{attribute 'qualified_only'}
VAR_GLOBAL
	senNO				: FB_Sensor_NO;
	senNC				: FB_Sensor_NC;
	senNO_2inRow		: FB_Sensor_NO_2InRow;
	
	senNO_TestDecorator			: FB_Sensor_NO_TestDecorator (fbToDecorate := senNO);
	senNC_TestDecorator			: FB_Sensor_NC_TestDecorator (fbToDecorate := senNC);
	senNO_2inRow_TestDecorator	: FB_Sensor_NO_2InRow_TestDecorator (fbToDecorate := senNO_2inRow);
	
END_VAR

(* stored: Version 1.1.0.1
   GVL GVL_Decorators: Id {93801117-c7f4-0fb3-1aa6-e6d5619250c7} *)
